{attribute 'qualified_only'}
{attribute 'strict'}
{attribute 'to_string'}
TYPE
ST110_Pnp_e :
(
    RESET := 0,         // Reset
	
    INIT := 100,        // Initialisieren 
    Init_VerticalUp_04 := 110,      // move axis below the mover to its rest position
    Init_VerticalUp_02_03 := 120,   // move the axis up to rest position
	Init_HomeHorizontals := 130,
	Init_HorizontalsToTrack := 140,
	Init_stop_vacum := 150,
	Init_check_if_pces_handled := 160,
	
    READY := 999,       // READY to Start, Init Done 
    START := 1000,      // Start Zyklisch
    MOVER_FREE_OP,      // Ab here, operation without mover can be done

	PnP_Hor_ToRotTablePos := 1010,
	PnP_WaitOnFeeder := 1020,
	PnP_Ver_RotTableDown := 1030,
	Vacum_on := 1040,
	PnP_Ver_RotTableUp := 1050,
	PnP_Hor_ToTrackPos := 1060,
    waitOnMover := 1070,        // wait until the mover is there
    MOVER_NEEDED_OP,    // Since here, a mover in position is needed to perform the action

	Pnp_Handling_pin_up := 1210,
	PnP_Ver_ShuttleDown := 1220,
	PnP_Ver_StartTorqueControl := 1225, // this step is used to start the execution of the movement
	                                    // even if the torque limit is passed. This way we ensure that
										// twincat motion library accept the move_absolute command
	PnP_Ver_ShuttleTorqueControl := 1230,
	PnP_Ver_quick_stop := 1240,
	Vacum_off := 1250,
	PnP_Ver_ShuttleUp := 1260,
	
    SYNC_MOVER_LEAVE,   // MoverMan need to take the mover
    DONE := 8000,       // Ablauf beendet 
    ERROR := 9000,      // Fehler 
    _max
);
END_TYPE

(* stored: Version 1.1.0.1, ProductVersion 3.1.4024.6
   EnumerationTextList ST110_Pnp_e: Id {34b51b03-fbba-42bb-849f-dbe203112bec} *)
